(* Logix 5000 project; controller EWEB_SOCK_UDP_VER2_2 1756-L63 rev 15.4; software revision 15.02 *)

TASK MainTask (periodic, rate 5 ms, priority 10, watchdog 500 ms) : MainProgram

MODULES
   Local : 1756-L63 (ICP 5, rev 15.4)
END_MODULES

TYPE READ_DATA_REQ :
STRUCT
   Timeout : DINT;
   BufLen : DINT;
END_STRUCT
END_TYPE

TYPE READ_RESP_DATA :
STRUCT
   FromAddr : SockAddr;
   BufLen : DINT;
   Buf : SINT[4096];
END_STRUCT
END_TYPE

TYPE REQUEST_PARAMETERS :
STRUCT
   Type : DINT;   // 1 -TCP, 2 - UDP
   Addr : SockAddr;
END_STRUCT
END_TYPE

TYPE SockAddr :
STRUCT
   Family : INT;   // Address Family Must be 2
   Port : INT;   // Port Number
   Addr : DINT;   // IP Address
END_STRUCT
END_TYPE

TYPE ST8 :
STRUCT
   LEN : DINT;
   DATA : SINT[8];
END_STRUCT
END_TYPE

TYPE STR_OUT :
STRUCT
   LEN : DINT;
   BUFF : SINT[480];
END_STRUCT
END_TYPE

TYPE Write_Data :
STRUCT
   Timeout : DINT;
   ToAddr : SockAddr;
   BufLen : DINT;
   Buf : SINT[20];
END_STRUCT
END_TYPE

TYPE WRT_DATA :
STRUCT
   Timeout : DINT;
   ToAddr : SockAddr;
   Buffer : STR_OUT;
END_STRUCT
END_TYPE

VAR_GLOBAL   (* controller tags *)
   _EWEB_PATH : STRING := '$01$07';
   _Local_Port : DINT := 10002;
   _Remote_IP_Addr : STRING := '100.100.90.254';
   _Remote_Port : DINT := 10001;
   Accept : ALIAS FOR Log_Enable.2;
   Attrubute : ALIAS FOR Log_Enable.6;
   Buf_LenSent : DINT := 7;
   Change_Log_MSG : MESSAGE;
        MessageParameters(ServiceCode := 16#0010, LocalElement := Log_Enable, ...)
   CLOCK : DINT[7] := ([0] := 1998, [1] := 1, [2] := 1, [4] := 4, [5] := 10, [6] := 993450);
   COLN : STRING := ':';
   Create : ALIAS FOR Log_Enable.0;
   Create_Sock_MSG : MESSAGE;
        MessageParameters(ServiceCode := 16#004b, LocalElement := SOCKET, DestinationTag := Instance, ...)
   Create_Socket_Request : BOOL;   // Manually Toggle This Bit to Create Socket
   Delete : ALIAS FOR Log_Enable.5;
   Delete_All_MSG : MESSAGE;
        MessageParameters(ServiceCode := 16#0051, ...)
   Delete_All_Request : BOOL;
   Delete_Sock_MSG : MESSAGE;
        MessageParameters(ServiceCode := 16#004f, ...)
   Delete_Sockets_Request : BOOL;   // Toggle This Bit to Delete Socket
   DOT : STRING := '.';
   dot_pos : DINT := 11;
   Errors : ALIAS FOR Log_Enable.7;
   Get_Sock_Instance_MSG : MESSAGE;
        MessageParameters(ServiceCode := 16#0001, DestinationTag := Socket_Instance_Data, ...)
   Get_Sock_Object_MSG : MESSAGE;
        MessageParameters(ServiceCode := 16#0001, DestinationTag := Socket_Object_Data, ...)
   Get_Socket_Instance_Request : BOOL;
   Get_Socket_Object_Request : BOOL;
   HOUR : STRING := '0';
   Instance : DINT := 13612;
   IP_A : STRING := '254';
   IP_A_D : DINT := 100;
   IP_B_D : DINT := 100;
   IP_C_D : DINT := 90;
   IP_D_D : DINT := 254;
   IP_DINT : DINT := 16#6464_5afe;
   ip_qty : DINT := 10;
   IP_st : DINT := 9;
   Log_Enable : DINT := 255;
   Log_old : DINT := 255;
   MINUTE : STRING := '04';
   Nothing : BOOL := 1;
   Open : ALIAS FOR Log_Enable.1;
   Read : ALIAS FOR Log_Enable.3;
   Read_Data_MSG : MESSAGE;
        MessageParameters(ServiceCode := 16#004d, LocalElement := Read_Data_Req, DestinationTag := Read_Response, ...)
   Read_Data_Req : READ_DATA_REQ := (Timeout := 1000, BufLen := 100);
   Read_Data_Request : BOOL;   // Toggle This Bit To Read Incoming Data
   Read_Response : READ_RESP_DATA := (FromAddr.Family := 2, FromAddr.Port := 10001, FromAddr.Addr := 1684298493, BufLen := 8, Buf[0] := 49, Buf[1] := 48, Buf[2] := 58, Buf[3] := 49, Buf[4] := 55, Buf[5] := 58, Buf[6] := 53, Buf[7] := 57, Buf[8] := 100, Buf[9] := 116, Buf[10] := 102, Buf[11] := 103, Buf[12] := 102, Buf[13] := 103, Buf[14] := 102, Buf[15] := 100, Buf[16] := 103, Buf[17] := 102, Buf[18] := 100, Buf[19] := 103, Buf[20] := 102, Buf[21] := 100, Buf[22] := 13, Buf[23] := 10, Buf[24] := 113, Buf[25] := 119, Buf[26] := 113, Buf[27] := 119, Buf[28] := 113, Buf[29] := 119, Buf[30] := 13, Buf[31] := 10, Buf[32] := 113, Buf[33] := 119, Buf[34] := 113, Buf[35] := 119, Buf[36] := 113, Buf[37] := 119, Buf[38] := 13, Buf[39] := 10);
   SECOND : STRING := '11';
   SOCKET : REQUEST_PARAMETERS := (Type := 2, Addr.Family := 2, Addr.Port := 10002);
   Socket_Instance_Data : DINT[13] := ([0] := 655425538, [4] := 2048, [5] := 2048, [6] := 8, [7] := 1, [8] := 300000);
   Socket_Object_Data : SINT[10];
   TIME : STRING := '0:04:10';
   Write : ALIAS FOR Log_Enable.4;
   Write_Data_MSG : MESSAGE;
        MessageParameters(ServiceCode := 16#004e, LocalElement := Write_Data_Out, DestinationTag := Buf_LenSent, ...)
   Write_Data_Out : WRT_DATA := (Timeout := 20000, ToAddr.Family := 2, ToAddr.Port := 10001, ToAddr.Addr := 1684298494, Buffer.LEN := 7, Buffer.BUFF[0] := 48, Buffer.BUFF[1] := 58, Buffer.BUFF[2] := 48, Buffer.BUFF[3] := 52, Buffer.BUFF[4] := 58, Buffer.BUFF[5] := 49, Buffer.BUFF[6] := 48, Buffer.BUFF[7] := 55, Buffer.BUFF[84] := 28, Buffer.BUFF[87] := -128, Buffer.BUFF[88] := 10, Buffer.BUFF[91] := -128, Buffer.BUFF[92] := 16, Buffer.BUFF[93] := 16, Buffer.BUFF[94] := -14, Buffer.BUFF[96] := 92, Buffer.BUFF[97] := 1, Buffer.BUFF[98] := 4, Buffer.BUFF[100] := -62, Buffer.BUFF[101] := 32, Buffer.BUFF[102] := 51, Buffer.BUFF[103] := -33, Buffer.BUFF[104] := 1, Buffer.BUFF[108] := 10, Buffer.BUFF[124] := 10, Buffer.BUFF[127] := -128, Buffer.BUFF[128] := 9, Buffer.BUFF[129] := 4, Buffer.BUFF[131] := -128, Buffer.BUFF[132] := 16, Buffer.BUFF[133] := 16, Buffer.BUFF[134] := -14, Buffer.BUFF[136] := 112, Buffer.BUFF[137] := 21, Buffer.BUFF[138] := 4, Buffer.BUFF[140] := -125, Buffer.BUFF[141] := -117, Buffer.BUFF[142] := -108, Buffer.BUFF[143] := -90, Buffer.BUFF[144] := 12, Buffer.BUFF[145] := 16, Buffer.BUFF[148] := 2, Buffer.BUFF[150] := 17, Buffer.BUFF[151] := 39, Buffer.BUFF[152] := -3, Buffer.BUFF[153] := 90, Buffer.BUFF[154] := 100, Buffer.BUFF[155] := 100, Buffer.BUFF[156] := 8, Buffer.BUFF[160] := 49, Buffer.BUFF[161] := 48, Buffer.BUFF[162] := 58, Buffer.BUFF[163] := 49, Buffer.BUFF[164] := 55, Buffer.BUFF[165] := 58,
        Buffer.BUFF[166] := 53, Buffer.BUFF[167] := 57, Buffer.BUFF[168] := 100, Buffer.BUFF[169] := 116, Buffer.BUFF[170] := 102, Buffer.BUFF[171] := 103, Buffer.BUFF[172] := 102, Buffer.BUFF[173] := 103, Buffer.BUFF[174] := 102, Buffer.BUFF[175] := 100, Buffer.BUFF[176] := 103, Buffer.BUFF[177] := 102, Buffer.BUFF[178] := 100, Buffer.BUFF[179] := 103, Buffer.BUFF[180] := 102, Buffer.BUFF[181] := 100, Buffer.BUFF[182] := 13, Buffer.BUFF[183] := 10, Buffer.BUFF[184] := 113, Buffer.BUFF[185] := 119, Buffer.BUFF[186] := 113, Buffer.BUFF[187] := 119, Buffer.BUFF[188] := 113, Buffer.BUFF[189] := 119, Buffer.BUFF[190] := 13, Buffer.BUFF[191] := 10, Buffer.BUFF[192] := 113, Buffer.BUFF[193] := 119, Buffer.BUFF[194] := 113, Buffer.BUFF[195] := 119, Buffer.BUFF[196] := 113, Buffer.BUFF[197] := 119, Buffer.BUFF[198] := 13, Buffer.BUFF[199] := 10);
   Write_Request : BOOL;   // Toggle This bit to Send Data Out
   zero : STRING := '0';
END_VAR

PROGRAM MainProgram   (* main routine _SOCKET_UDP *)

ROUTINE _SOCKET_STATS   (* ladder *)
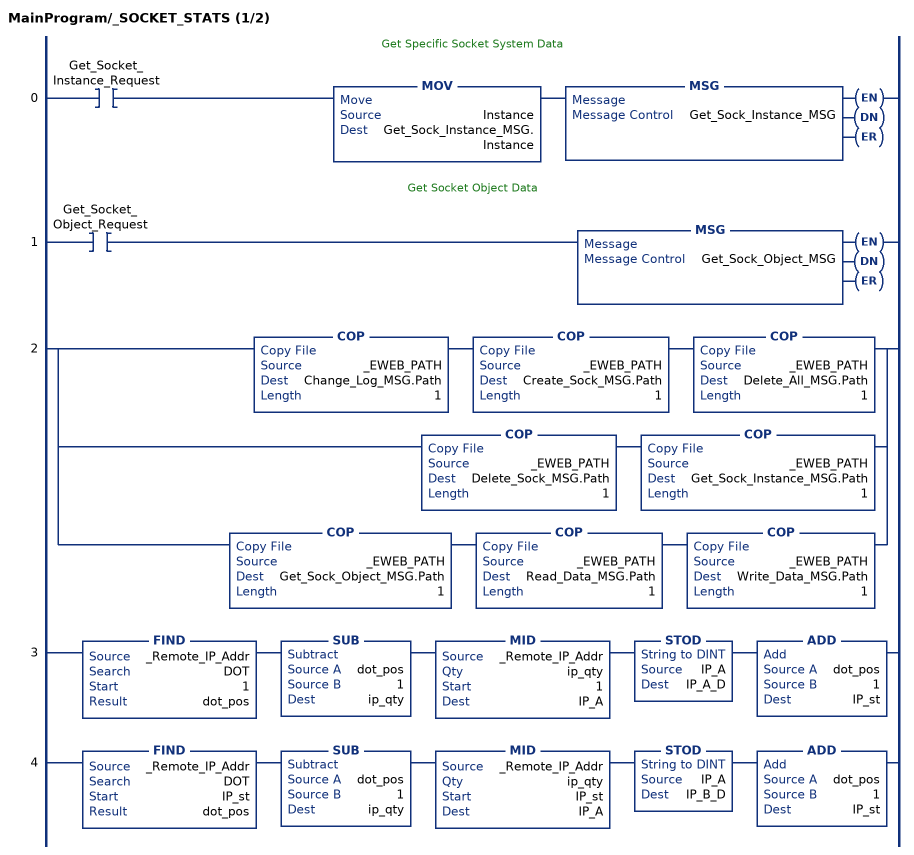
   // Get Specific Socket System Data
   0: XIC(Get_Socket_Instance_Request)MOV(Instance,Get_Sock_Instance_MSG.Instance)MSG(Get_Sock_Instance_MSG);
   // Get Socket Object Data
   1: XIC(Get_Socket_Object_Request)MSG(Get_Sock_Object_MSG);
   2: [COP(_EWEB_PATH,Change_Log_MSG.Path,1) COP(_EWEB_PATH,Create_Sock_MSG.Path,1) COP(_EWEB_PATH,Delete_All_MSG.Path,1) ,COP(_EWEB_PATH,Delete_Sock_MSG.Path,1) COP(_EWEB_PATH,Get_Sock_Instance_MSG.Path,1) ,COP(_EWEB_PATH,Get_Sock_Object_MSG.Path,1) COP(_EWEB_PATH,Read_Data_MSG.Path,1) COP(_EWEB_PATH,Write_Data_MSG.Path,1) ];
   3: FIND(_Remote_IP_Addr,DOT,1,dot_pos)SUB(dot_pos,1,ip_qty)MID(_Remote_IP_Addr,ip_qty,1,IP_A)STOD(IP_A,IP_A_D)ADD(dot_pos,1,IP_st);
   4: FIND(_Remote_IP_Addr,DOT,IP_st,dot_pos)SUB(dot_pos,1,ip_qty)MID(_Remote_IP_Addr,ip_qty,IP_st,IP_A)STOD(IP_A,IP_B_D)ADD(dot_pos,1,IP_st);
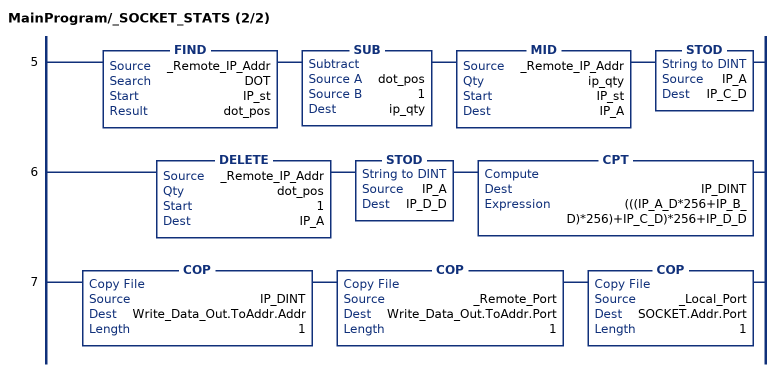
   5: FIND(_Remote_IP_Addr,DOT,IP_st,dot_pos)SUB(dot_pos,1,ip_qty)MID(_Remote_IP_Addr,ip_qty,IP_st,IP_A)STOD(IP_A,IP_C_D);
   6: DELETE(_Remote_IP_Addr,dot_pos,1,IP_A)STOD(IP_A,IP_D_D)CPT(IP_DINT,(((IP_A_D*256+IP_B_D)*256)+IP_C_D)*256+IP_D_D);
   7: COP(IP_DINT,Write_Data_Out.ToAddr.Addr,1)COP(_Remote_Port,Write_Data_Out.ToAddr.Port,1)COP(_Local_Port,SOCKET.Addr.Port,1);
END_ROUTINE

ROUTINE _SOCKET_UDP   (* ladder *)
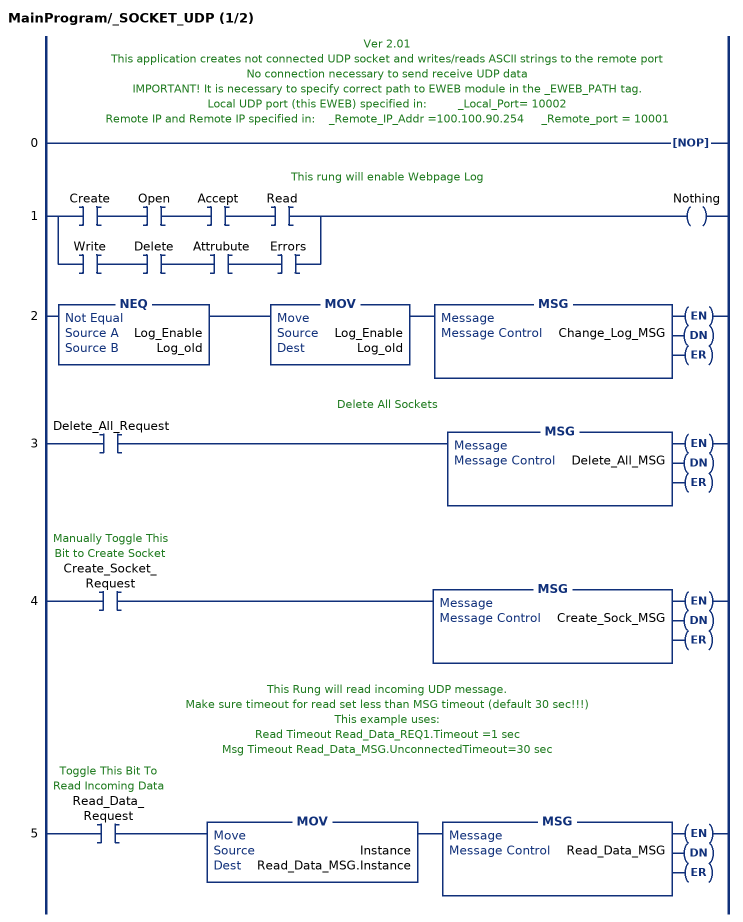
   // Ver 2.01
   // This application creates not connected UDP socket and writes/reads ASCII strings to the remote port
   // No connection necessary to send receive UDP data
   // IMPORTANT! It is necessary to specify correct path to EWEB module in the _EWEB_PATH tag.
   // Local UDP port (this EWEB) specified in:         _Local_Port= 10002
   // Remote IP and Remote IP specified in:    _Remote_IP_Addr =100.100.90.254     _Remote_port = 10001
   0: NOP();
   // This rung will enable Webpage Log
   1: [XIC(Create) XIC(Open) XIC(Accept) XIC(Read) ,XIC(Write) XIC(Delete) XIC(Attrubute) XIC(Errors) ]OTE(Nothing);
   2: NEQ(Log_Enable,Log_old)MOV(Log_Enable,Log_old)MSG(Change_Log_MSG);
   // Delete All Sockets
   3: XIC(Delete_All_Request)MSG(Delete_All_MSG);
   4: XIC(Create_Socket_Request)MSG(Create_Sock_MSG);
   // This Rung will read incoming UDP message.
   // Make sure timeout for read set less than MSG timeout (default 30 sec!!!)
   // This example uses:
   // Read Timeout Read_Data_REQ1.Timeout =1 sec
   // Msg Timeout Read_Data_MSG.UnconnectedTimeout=30 sec
   5: XIC(Read_Data_Request)MOV(Instance,Read_Data_MSG.Instance)MSG(Read_Data_MSG);
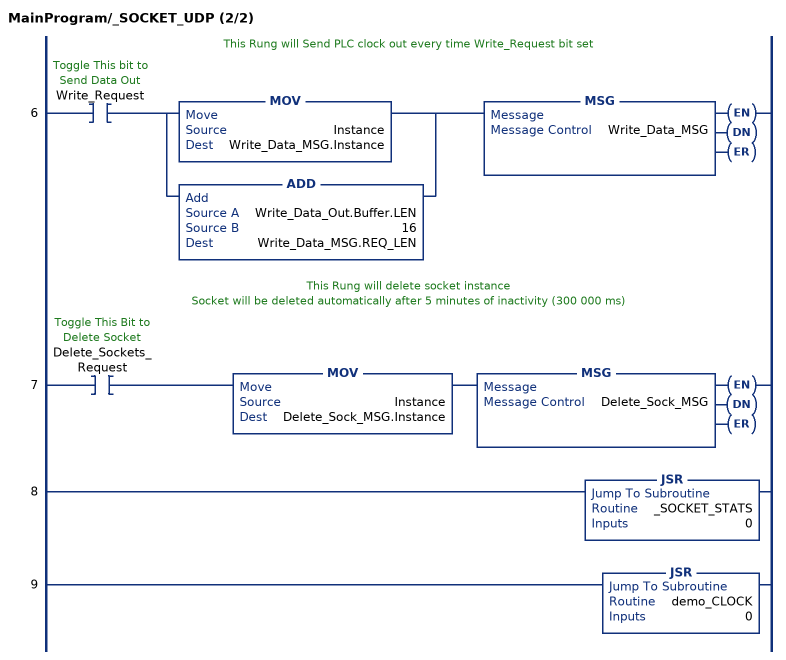
   // This Rung will Send PLC clock out every time Write_Request bit set
   6: XIC(Write_Request)[MOV(Instance,Write_Data_MSG.Instance) ,ADD(Write_Data_Out.Buffer.LEN,16,Write_Data_MSG.REQ_LEN) ]MSG(Write_Data_MSG);
   // This Rung will delete socket instance
   // Socket will be deleted automatically after 5 minutes of inactivity (300 000 ms)
   7: XIC(Delete_Sockets_Request)MOV(Instance,Delete_Sock_MSG.Instance)MSG(Delete_Sock_MSG);
   8: JSR(_SOCKET_STATS,0);
   9: JSR(demo_CLOCK,0);
END_ROUTINE

ROUTINE demo_CLOCK   (* ladder *)
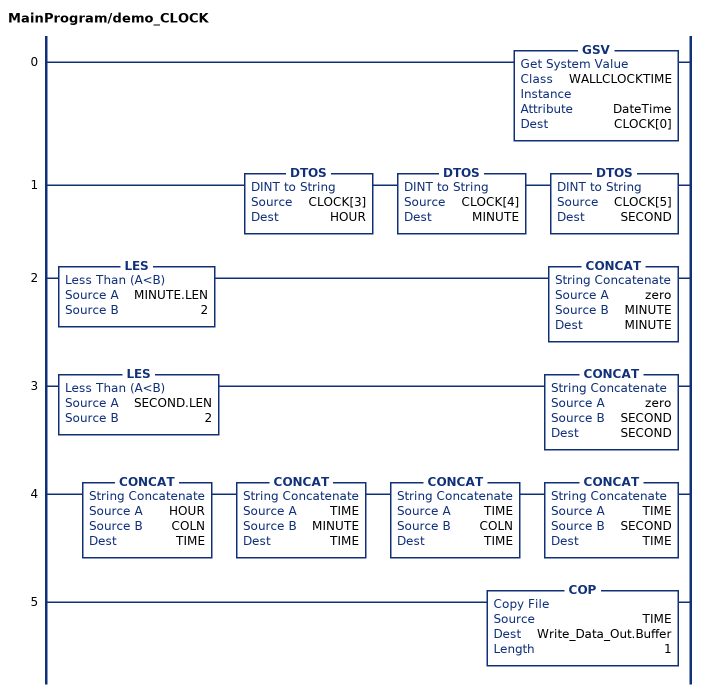
   0: GSV(WALLCLOCKTIME,,DateTime,CLOCK[0]);
   1: DTOS(CLOCK[3],HOUR)DTOS(CLOCK[4],MINUTE)DTOS(CLOCK[5],SECOND);
   2: LES(MINUTE.LEN,2)CONCAT(zero,MINUTE,MINUTE);
   3: LES(SECOND.LEN,2)CONCAT(zero,SECOND,SECOND);
   4: CONCAT(HOUR,COLN,TIME)CONCAT(TIME,MINUTE,TIME)CONCAT(TIME,COLN,TIME)CONCAT(TIME,SECOND,TIME);
   5: COP(TIME,Write_Data_Out.Buffer,1);
END_ROUTINE
END_PROGRAM
